{attribute addProperty BoxType "EL3058-0000-0017"}
{attribute addProperty Id "AI_Standard_ChannelAT %I*ARRAY[0..14] OF AI_Standard_Channel_B51B79FC648810WcStateAT %I*WcState_98A4DF7520.250InfoDataAT %I*InfoData_BC63D37F80100"}
{attribute addProperty CRC "3084020167"}
{attribute addProperty SizeInBites "730"}
{attribute addProperty SizeInBytes "91.25"}
TYPE EL3058_6F92BA30 :
STRUCT
	{attribute addProperty Name "AI_Standard_Channel"}
	AI_Standard_Channel : ARRAY[0..14] OF AI_Standard_Channel_B51B79FC;
	{attribute addProperty Name "WcState"}
	WcState : WcState_98A4DF75;
	{attribute addProperty Name "InfoData"}
	InfoData : InfoData_BC63D37F;
END_STRUCT
END_TYPE

(* stored: Version 1.2.0.0, ProductVersion 3.1.4024.9
   DUT EL3058_6F92BA30: Id {d2248de8-366f-4a33-a4ca-75e674b4bed7} *)
